   // Определение аварий и предупреждений для отображения на HMI
   // PCV300
   IF "REG_Data".PCV300_Message.Error OR "REG_Data".PCV300_Message.Term_error OR
       "REG_Data".PCV300_Message.Phase_failure OR "REG_Data".PCV300_Status.Error OR
       "REG_Data".PCV300_Status.Fail OR "REG_Master".PCV300_error
   THEN
       "Regs".PCV300_Alarm := true;
   ELSE
       "Regs".PCV300_Alarm := false;
   END_IF;

   IF "REG_Data".PCV300_Message.Warning OR "REG_Data".PCV300_Status.Warning
   THEN
       "Regs".PCV300_Warning := true;
   ELSE
       "Regs".PCV300_Warning := false;
   END_IF;

   // LCV300
   IF "REG_Data".LCV300_Message.Error OR "REG_Data".LCV300_Message.Term_error OR
       "REG_Data".LCV300_Message.Phase_failure OR "REG_Data".LCV300_Status.Error OR
       "REG_Data".LCV300_Status.Fail OR "REG_Master".LCV300_error
   THEN
       "Regs".LCV300_Alarm := true;
   ELSE
       "Regs".LCV300_Alarm := false;
   END_IF;

   IF "REG_Data".LCV300_Message.Warning OR "REG_Data".LCV300_Status.Warning
   THEN
       "Regs".LCV300_Warning := true;
   ELSE
       "Regs".LCV300_Warning := false;
   END_IF;
END_FUNCTION

FUNCTION "Modbus_init" : Void   // FC11, SCL
{ S7_Optimized_Access := 'TRUE' }
VERSION : 0.1
BEGIN
   //************************************************ Регуляторы *****************************************************************
   "PortSettings".Regs."Port" := 258;
   "PortSettings".Regs.Baud := 19200;
   "PortSettings".Regs.Parity := 0;
   "REG_Master".Settings.MB_Addr := 1;
   "REG_Master".State := 10;

   "REG_Master".reqREGmaster := 0;
   "Modbus_Comm_Load_Regs".MODE := 4; // Operating mode 4 = Half duplex (RS485) two-wire mode
   "Modbus_Comm_Load_Regs"(REQ := true,
                           "PORT" := "PortSettings".Regs."Port",
                           BAUD := "PortSettings".Regs.Baud,
                           PARITY := "PortSettings".Regs.Parity,
                           FLOW_CTRL := 0,
                           RTS_ON_DLY := 0,
                           RTS_OFF_DLY := 0,
                           RESP_TO := 1000,
                           DONE => "PortSettings".Regs.Done,
                           ERROR => "PortSettings".Regs.Error,
                           STATUS => "PortSettings".Regs.Status,
                           MB_DB := "Modbus_Master_Regs".MB_DB);

   //************************************************ Передача на верхний уровень **************************************************
   "PortSettings".Up."Port" := 257;
   "PortSettings".Up.Baud := 9600;
   "PortSettings".Up.Parity := 0;

   "Modbus_Comm_Load_Up".MODE := 4; // Operating mode 4 = Half duplex (RS485) two-wire mode
   "Modbus_Comm_Load_Up"(REQ := true,
                         "PORT" := "PortSettings".Up."Port",
                         BAUD := "PortSettings".Up.Baud,
                         PARITY := "PortSettings".Up.Parity,
                         FLOW_CTRL := 0,
                         RTS_ON_DLY := 0,
                         RTS_OFF_DLY := 0,
                         RESP_TO := 1000,
                         DONE => "PortSettings".Up.Done,
                         ERROR => "PortSettings".Up.Error,
                         STATUS => "PortSettings".Up.Status,
                         MB_DB := "Modbus_Slave_Up".MB_DB);

   //************************************************ УВП **************************************************
   "MB_CLIENT_UVP".MB_Unit_ID := 1;
   "MB_CLIENT_UVP".MB_Transaction_ID := 1;
   "UVP_States".Connect_UVP.InterfaceId := 64;
   "UVP_States".Connect_UVP.ID := 1;
   "UVP_States".Connect_UVP.ActiveEstablished := true;
   "UVP_States".Connect_UVP.RemoteAddress.ADDR[1] := 10;
   "UVP_States".Connect_UVP.RemoteAddress.ADDR[2] := 158;
   "UVP_States".Connect_UVP.RemoteAddress.ADDR[3] := 144;
   "UVP_States".Connect_UVP.RemoteAddress.ADDR[4] := 30;
   "UVP_States".Connect_UVP.RemotePort := 502;
END_FUNCTION

FUNCTION "DATA_FC" : Void   // FC14, SCL
{ S7_Optimized_Access := 'TRUE' }
VERSION : 0.1
BEGIN
   // Перекладка данных в DATA

    "DATA".Measuring.PT100_Value := "PT100".Signal_AI.Value;
    "DATA".Measuring.PT100_Circuit := "PT100".Signal_AI.Circuit;
    "DATA".Measuring.TT100_Value := "TT100".Signal_AI.Value;
    "DATA".Measuring.TT100_Circuit := "TT100".Signal_AI.Circuit;
    "DATA".Measuring.LT100_Value := "LT100".Signal_AI.Value;
    "DATA".Measuring.LT100_Circuit := "LT100".Signal_AI.Circuit;
    "DATA".Measuring.AG100_Value := "AG100".Signal_AI.Value;
    "DATA".Measuring. AG100_Circuit := "AG100".Signal_AI.Circuit;
    "DATA".Measuring.PT200_Value := "PT200".Signal_AI.Value;
    "DATA".Measuring.PT200_Circuit := "PT200".Signal_AI.Circuit;
    "DATA".Measuring.TT200_Value := "TT200".Signal_AI.Value;
    "DATA".Measuring.TT200_Circuit := "TT200".Signal_AI.Circuit;
    "DATA".Measuring.LT200_Value := "LT200".Signal_AI.Value;
    "DATA".Measuring.LT200_Circuit := "LT200".Signal_AI.Circuit;
    "DATA".Measuring.AG200_Value := "AG200".Signal_AI.Value;
    "DATA".Measuring.AG200_Circuit := "AG200".Signal_AI.Circuit;
    "DATA".Measuring.TT500_Value := "TT500".Signal_AI.Value;
    "DATA".Measuring.TT500_Circuit := "TT500".Signal_AI.Circuit;
    "DATA".Measuring.PCV300_Pologenie := "REG_Data".PCV300_Pologenie_ok;
    "DATA".Measuring.LCV300_Pologenie := "REG_Data".LCV300_Pologenie_ok;
    //
    "DATA".Measuring.SIKG_Press := "UVP_Data".UVP1_Current_L1.UVP_Press;
    "DATA".Measuring.SIKG_Temp := "UVP_Data".UVP1_Current_L1.UVP_Temp;
    "DATA".Measuring.SIKG_Flow_ru := "UVP_Data".UVP1_Current_L1.UVP_vol_flow_work;
    "DATA".Measuring.SIKG_Flow_stu := "UVP_Data".UVP1_Current_L1.UVP_vol_flow_norm;
    "DATA".Measuring.SIKG_Flow_ru_prev2h := "UVP_Data".UVP1_Cumulative_L1.UVP_Vol_work_prev2h;
    "DATA".Measuring.SIKG_Flow_stu_prev2h := "UVP_Data".UVP1_Cumulative_L1.UVP_Vol_norm_prev2h;
    "DATA".Measuring.SIKG_Flow_ru_prevDay := "UVP_Data".UVP1_Cumulative_L1.UVP_Vol_work_prevDay;
    "DATA".Measuring.SIKG_Flow_stu_prevDay := "UVP_Data".UVP1_Cumulative_L1.UVP_Vol_norm_prevDay;
    "DATA".Measuring.SIKG_total := "UVP_Data".UVP1_Current_L1.UVP_Vol_norm;
    //
    "DATA".Measuring.SIKN_MassFlow := "UVP_Data".UVP1_Current_L2.UVP_Param_vol_flow_work;
    "DATA".Measuring.SIKN_MassFlow_prev2h := "UVP_Data".UVP1_Cumulative_L2.UVP_Param_vol_flow_work_prev2h;
    "DATA".Measuring.SIKN_MassFlow_prevDay := "UVP_Data".UVP1_Cumulative_L2.UVP_Param_vol_flow_work_prevDay;
    "DATA".Measuring.SIKN_total := "UVP_Data".UVP1_Current_L2.UVP_Vol_work;

    // ***************************** СТАТУСЫ УСТРОЙСТВ *********************************
    // Статус XV100
    IF ("DI3".Slot.Pins[6] OR "DATA".Measuring.XV100_no_cmd_close OR "DATA".Measuring.XV100_no_cmd_open) THEN
        "DATA".Measuring.XV100_State := 3; // Авария
    ELSIF ("DI3".Slot.Pins[4] AND NOT "DI3".Slot.Pins[5]) THEN
        "DATA".Measuring.XV100_State := 2; // Открыт
    ELSIF ("DI3".Slot.Pins[5] AND NOT "DI3".Slot.Pins[4]) THEN
        "DATA".Measuring.XV100_State := 1; // Закрыт
    ELSE
        "DATA".Measuring.XV100_State := 0; // Неопределено
    END_IF;

    // Статус обогрева
    IF ("Head".Device.Fail > 0) THEN
        "DATA".Measuring.Head_State := 2; // Авария
    ELSIF ("Head".Device.State = 1) THEN
        "DATA".Measuring.Head_State := 1; // Включен
    ELSIF ("Head".Device.State = 0) THEN
        "DATA".Measuring.Head_State := 0; // Выключен
    END_IF;

    // Статус питания установки
    IF ("Power".Device.Fail > 0) THEN
        "DATA".Measuring.Power_State := 2; // Авария
    ELSIF ("Power".Device.State = 1) THEN
        "DATA".Measuring.Power_State := 1; // Включен
    ELSIF ("Power".Device.State = 0) THEN
        "DATA".Measuring.Power_State := 0; // Выключен
    END_IF;

    "DATA".Measuring.PCV300_Alarm := "Regs".PCV300_Alarm;
    "DATA".Measuring.PCV300_Warning := "Regs".PCV300_Warning;
    "DATA".Measuring.PCV300_Midle := "Regs".PCV300_Midle;
    "DATA".Measuring.PCV300_DIST := "REG_Data".PCV300_Message.Selector_DIST;
    "DATA".Measuring.PCV300_LOCAL := "REG_Data".PCV300_Message.Selector_LOCAL;
    "DATA".Measuring.LCV300_Alarm := "Regs".LCV300_Alarm;
    "DATA".Measuring.LCV300_Warning := "Regs".LCV300_Warning;
    "DATA".Measuring.LCV300_Midle := "Regs".LCV300_Midle;
    "DATA".Measuring.LCV300_DIST := "REG_Data".LCV300_Message.Selector_DIST;
    "DATA".Measuring.LCV300_LOCAL := "REG_Data".LCV300_Message.Selector_LOCAL;
    "DATA".Measuring.LS100 := "DI1".Slot.Pins[0];
    "DATA".Measuring.LS101 := "DI1".Slot.Pins[2];
    "DATA".Measuring.LS200 := "DI1".Slot.Pins[4];
    "DATA".Measuring.LS201 := "DI1".Slot.Pins[6];
    "DATA".Measuring.HS600_Emer_stop := "DI2".Slot.Pins[3];
    "DATA".Measuring.Head_run := "DI2".Slot.Pins[7];
    "DATA".Measuring.Power_run := "DI2".Slot.Pins[6];
    "DATA".Measuring.XV100_open := "DI3".Slot.Pins[4];
    "DATA".Measuring.XV100_close := "DI3".Slot.Pins[5];
    "DATA".Measuring.XV100_fault := "DI3".Slot.Pins[6];
    "DATA".Measuring.Spark := "DO1".Slot.Pins[4];

    "DATA".Measuring.PT100_HH_Alarm := "PT100".Signal_AI.HH_Alarm;
    "DATA".Measuring.PT100_H_Alarm := "PT100".Signal_AI.H_Alarm;
    "DATA".Measuring.PT100_L_Alarm := "PT100".Signal_AI.L_Alarm;
    "DATA".Measuring.PT100_LL_Alarm := "PT100".Signal_AI.LL_Alarm;
    "DATA".Measuring.PT100_Chan_Fail := "PT100".Signal_AI.Chan_Fail;
    "DATA".Measuring.PT100_Sim := "PT100".Signal_AI.Sim_En;

    "DATA".Measuring.TT100_HH_Alarm := "TT100".Signal_AI.HH_Alarm;
    "DATA".Measuring.TT100_H_Alarm := "TT100".Signal_AI.H_Alarm;
    "DATA".Measuring.TT100_L_Alarm := "TT100".Signal_AI.L_Alarm;
    "DATA".Measuring.TT100_LL_Alarm := "TT100".Signal_AI.LL_Alarm;
    "DATA".Measuring.TT100_Chan_Fail := "TT100".Signal_AI.Chan_Fail;
    "DATA".Measuring.TT100_Sim := "TT100".Signal_AI.Sim_En;

    "DATA".Measuring.LT100_HH_Alarm := "LT100".Signal_AI.HH_Alarm;
    "DATA".Measuring.LT100_H_Alarm := "LT100".Signal_AI.H_Alarm;
    "DATA".Measuring.LT100_L_Alarm := "LT100".Signal_AI.L_Alarm;
    "DATA".Measuring.LT100_LL_Alarm := "LT100".Signal_AI.LL_Alarm;
    "DATA".Measuring.LT100_Chan_Fail := "LT100".Signal_AI.Chan_Fail;
    "DATA".Measuring.LT100_Sim := "LT100".Signal_AI.Sim_En;

    "DATA".Measuring.AG100_HH_Alarm := "AG100".Signal_AI.HH_Alarm;
    "DATA".Measuring.AG100_H_Alarm := "AG100".Signal_AI.H_Alarm;
    "DATA".Measuring.AG100_L_Alarm := "AG100".Signal_AI.L_Alarm;
    "DATA".Measuring.AG100_LL_Alarm := "AG100".Signal_AI.LL_Alarm;
    "DATA".Measuring.AG100_Chan_Fail := "AG100".Signal_AI.Chan_Fail;
    "DATA".Measuring.AG100_Sim := "AG100".Signal_AI.Sim_En;

    "DATA".Measuring.PT200_HH_Alarm := "PT200".Signal_AI.HH_Alarm;
    "DATA".Measuring.PT200_H_Alarm := "PT200".Signal_AI.H_Alarm;
    "DATA".Measuring.PT200_L_Alarm := "PT200".Signal_AI.L_Alarm;
    "DATA".Measuring.PT200_LL_Alarm := "PT200".Signal_AI.LL_Alarm;
    "DATA".Measuring.PT200_Chan_Fail := "PT200".Signal_AI.Chan_Fail;
    "DATA".Measuring.PT200_Sim := "PT200".Signal_AI.Sim_En;

    "DATA".Measuring.TT200_HH_Alarm := "TT200".Signal_AI.HH_Alarm;
    "DATA".Measuring.TT200_H_Alarm := "TT200".Signal_AI.H_Alarm;
    "DATA".Measuring.TT200_L_Alarm := "TT200".Signal_AI.L_Alarm;
    "DATA".Measuring.TT200_LL_Alarm := "TT200".Signal_AI.LL_Alarm;
    "DATA".Measuring.TT200_Chan_Fail := "TT200".Signal_AI.Chan_Fail;
    "DATA".Measuring.TT200_Sim := "TT200".Signal_AI.Sim_En;

    "DATA".Measuring.LT200_HH_Alarm := "LT200".Signal_AI.HH_Alarm;
    "DATA".Measuring.LT200_H_Alarm := "LT200".Signal_AI.H_Alarm;
    "DATA".Measuring.LT200_L_Alarm := "LT200".Signal_AI.L_Alarm;
    "DATA".Measuring.LT200_LL_Alarm := "LT200".Signal_AI.LL_Alarm;
    "DATA".Measuring.LT200_Chan_Fail := "LT200".Signal_AI.Chan_Fail;
    "DATA".Measuring.LT200_Sim := "LT200".Signal_AI.Sim_En;

    "DATA".Measuring.AG200_HH_Alarm := "AG200".Signal_AI.HH_Alarm;
    "DATA".Measuring.AG200_H_Alarm := "AG200".Signal_AI.H_Alarm;
    "DATA".Measuring.AG200_L_Alarm := "AG200".Signal_AI.L_Alarm;
    "DATA".Measuring.AG200_LL_Alarm := "AG200".Signal_AI.LL_Alarm;
    "DATA".Measuring.AG200_Chan_Fail := "AG200".Signal_AI.Chan_Fail;
    "DATA".Measuring.AG200_Sim := "AG200".Signal_AI.Sim_En;

    "DATA".Measuring.TT500_HH_Alarm := "TT500".Signal_AI.HH_Alarm;
    "DATA".Measuring.TT500_H_Alarm := "TT500".Signal_AI.H_Alarm;
    "DATA".Measuring.TT500_L_Alarm := "TT500".Signal_AI.L_Alarm;
    "DATA".Measuring.TT500_LL_Alarm := "TT500".Signal_AI.LL_Alarm;
    "DATA".Measuring.TT500_Chan_Fail := "TT500".Signal_AI.Chan_Fail;
    "DATA".Measuring.TT500_Sim := "TT500".Signal_AI.Sim_En;



   // Запись команд из DATA
    "PT100".Signal_AI.Scal_Max_Eu := "DATA".Commands.PT100_Scal_Max_Eu;
    "PT100".Signal_AI.Scal_Min_Eu := "DATA".Commands.PT100_Scal_Min_Eu;
    "PT100".Signal_AI.HH_Lim := "DATA".Commands.PT100_HH_Lim;
    "PT100".Signal_AI.H_Lim := "DATA".Commands.PT100_H_Lim;
    "PT100".Signal_AI.L_Lim := "DATA".Commands.PT100_L_Lim;
    "PT100".Signal_AI.LL_Lim := "DATA".Commands.PT100_LL_Lim;
    "PT100".Signal_AI.Sim_Value := "DATA".Commands.PT100_Sim_Value;

    "TT100".Signal_AI.Scal_Max_Eu := "DATA".Commands.TT100_Scal_Max_Eu;
    "TT100".Signal_AI.Scal_Min_Eu := "DATA".Commands.TT100_Scal_Min_Eu;
    "TT100".Signal_AI.HH_Lim := "DATA".Commands.TT100_HH_Lim;
    "TT100".Signal_AI.H_Lim := "DATA".Commands.TT100_H_Lim;
    "TT100".Signal_AI.L_Lim := "DATA".Commands.TT100_L_Lim;
    "TT100".Signal_AI.LL_Lim := "DATA".Commands.TT100_LL_Lim;
    "TT100".Signal_AI.Sim_Value := "DATA".Commands.TT100_Sim_Value;

    "LT100".Signal_AI.Scal_Max_Eu := "DATA".Commands.LT100_Scal_Max_Eu;
    "LT100".Signal_AI.Scal_Min_Eu := "DATA".Commands.LT100_Scal_Min_Eu;
    "LT100".Signal_AI.HH_Lim := "DATA".Commands.LT100_HH_Lim;
    "LT100".Signal_AI.H_Lim := "DATA".Commands.LT100_H_Lim;
    "LT100".Signal_AI.L_Lim := "DATA".Commands.LT100_L_Lim;
    "LT100".Signal_AI.LL_Lim := "DATA".Commands.LT100_LL_Lim;
    "LT100".Signal_AI.Sim_Value := "DATA".Commands.LT100_Sim_Value;

    "AG100".Signal_AI.Scal_Max_Eu := "DATA".Commands.AG100_Scal_Max_Eu;
    "AG100".Signal_AI.Scal_Min_Eu := "DATA".Commands.AG100_Scal_Min_Eu;
    "AG100".Signal_AI.HH_Lim := "DATA".Commands.AG100_HH_Lim;
    "AG100".Signal_AI.H_Lim := "DATA".Commands.AG100_H_Lim;
    "AG100".Signal_AI.L_Lim := "DATA".Commands.AG100_L_Lim;
    "AG100".Signal_AI.LL_Lim := "DATA".Commands.AG100_LL_Lim;
    "AG100".Signal_AI.Sim_Value := "DATA".Commands.AG100_Sim_Value;

    "PT200".Signal_AI.Scal_Max_Eu := "DATA".Commands.PT200_Scal_Max_Eu;
    "PT200".Signal_AI.Scal_Min_Eu := "DATA".Commands.PT200_Scal_Min_Eu;
    "PT200".Signal_AI.HH_Lim := "DATA".Commands.PT200_HH_Lim;
    "PT200".Signal_AI.H_Lim := "DATA".Commands.PT200_H_Lim;
    "PT200".Signal_AI.L_Lim := "DATA".Commands.PT200_L_Lim;
    "PT200".Signal_AI.LL_Lim := "DATA".Commands.PT200_LL_Lim;
    "PT200".Signal_AI.Sim_Value := "DATA".Commands.PT200_Sim_Value;

    "TT200".Signal_AI.Scal_Max_Eu := "DATA".Commands.TT200_Scal_Max_Eu;
    "TT200".Signal_AI.Scal_Min_Eu := "DATA".Commands.TT200_Scal_Min_Eu;
    "TT200".Signal_AI.HH_Lim := "DATA".Commands.TT200_HH_Lim;
    "TT200".Signal_AI.H_Lim := "DATA".Commands.TT200_H_Lim;
    "TT200".Signal_AI.L_Lim := "DATA".Commands.TT200_L_Lim;
    "TT200".Signal_AI.LL_Lim := "DATA".Commands.TT200_LL_Lim;
    "TT200".Signal_AI.Sim_Value := "DATA".Commands.TT200_Sim_Value;

    "LT200".Signal_AI.Scal_Max_Eu := "DATA".Commands.LT200_Scal_Max_Eu;
    "LT200".Signal_AI.Scal_Min_Eu := "DATA".Commands.LT200_Scal_Min_Eu;
    "LT200".Signal_AI.HH_Lim := "DATA".Commands.LT200_HH_Lim;
    "LT200".Signal_AI.H_Lim := "DATA".Commands.LT200_H_Lim;
    "LT200".Signal_AI.L_Lim := "DATA".Commands.LT200_L_Lim;
    "LT200".Signal_AI.LL_Lim := "DATA".Commands.LT200_LL_Lim;
    "LT200".Signal_AI.Sim_Value := "DATA".Commands.LT200_Sim_Value;

    "AG200".Signal_AI.Scal_Max_Eu := "DATA".Commands.AG200_Scal_Max_Eu;
    "AG200".Signal_AI.Scal_Min_Eu := "DATA".Commands.AG200_Scal_Min_Eu;
    "AG200".Signal_AI.HH_Lim := "DATA".Commands.AG200_HH_Lim;
    "AG200".Signal_AI.H_Lim := "DATA".Commands.AG200_H_Lim;
    "AG200".Signal_AI.L_Lim := "DATA".Commands.AG200_L_Lim;
    "AG200".Signal_AI.LL_Lim := "DATA".Commands.AG200_LL_Lim;
    "AG200".Signal_AI.Sim_Value := "DATA".Commands.AG200_Sim_Value;

    "TT500".Signal_AI.Scal_Max_Eu := "DATA".Commands.TT500_Scal_Max_Eu;
    "TT500".Signal_AI.Scal_Min_Eu := "DATA".Commands.TT500_Scal_Min_Eu;
    "TT500".Signal_AI.HH_Lim := "DATA".Commands.TT500_HH_Lim;
    "TT500".Signal_AI.H_Lim := "DATA".Commands.TT500_H_Lim;
    "TT500".Signal_AI.L_Lim := "DATA".Commands.TT500_L_Lim;
    "TT500".Signal_AI.LL_Lim := "DATA".Commands.TT500_LL_Lim;
    "TT500".Signal_AI.Sim_Value := "DATA".Commands.TT500_Sim_Value;

    "PCV300".Setpoint := "DATA".Commands.PCV300_Setpoint;
    "PCV300".ManualValue := "DATA".Commands.PCV300_ManualValue;
    "PCV300".Retain.CtrlParams.Gain := "DATA".Commands.PCV300_Gain;
    "PCV300".Retain.CtrlParams.Ti := "DATA".Commands.PCV300_Ti;
    "PCV300".Retain.CtrlParams.Td := "DATA".Commands.PCV300_Td;
    "PCV300".Retain.CtrlParams.TdFiltRatio := "DATA".Commands.PCV300_TdFiltRatio;
    "PCV300".Config.OutputUpperLimit := "DATA".Commands.PCV300_OutputUpperLimit;
    "PCV300".Config.OutputLowerLimit := "DATA".Commands.PCV300_OutputLowerLimit;

    "LCV300".Setpoint := "DATA".Commands. LCV300_Setpoint;
    "LCV300".ManualValue := "DATA".Commands. LCV300_ManualValue;
    "LCV300".Retain.CtrlParams.Gain := "DATA".Commands. LCV300_Gain;
    "LCV300".Retain.CtrlParams.Ti := "DATA".Commands. LCV300_Ti;
    "LCV300".Retain.CtrlParams.Td := "DATA".Commands. LCV300_Td;
    "LCV300".Retain.CtrlParams.TdFiltRatio := "DATA".Commands. LCV300_TdFiltRatio;
    "LCV300".Config.OutputUpperLimit := "DATA".Commands. LCV300_OutputUpperLimit;
    "LCV300".Config.OutputLowerLimit := "DATA".Commands. LCV300_OutputLowerLimit;

    "PT100".Signal_AI.HH_Alarm_En := "DATA".Commands.PT100_HH_Alarm_En;
    "PT100".Signal_AI.H_Alarm_En := "DATA".Commands.PT100_H_Alarm_En;
    "PT100".Signal_AI.L_Alarm_En := "DATA".Commands.PT100_L_Alarm_En;
    "PT100".Signal_AI.LL_Alarm_En := "DATA".Commands.PT100_LL_Alarm_En;
    "PT100".Signal_AI.Sim_En := "DATA".Commands.PT100_Sim_En;

    "TT100".Signal_AI.HH_Alarm_En := "DATA".Commands.TT100_HH_Alarm_En;
    "TT100".Signal_AI.H_Alarm_En := "DATA".Commands.TT100_H_Alarm_En;
    "TT100".Signal_AI.L_Alarm_En := "DATA".Commands.TT100_L_Alarm_En;
    "TT100".Signal_AI.LL_Alarm_En := "DATA".Commands.TT100_LL_Alarm_En;
    "TT100".Signal_AI.Sim_En := "DATA".Commands.TT100_Sim_En;

    "LT100".Signal_AI.HH_Alarm_En := "DATA".Commands.LT100_HH_Alarm_En;
    "LT100".Signal_AI.H_Alarm_En := "DATA".Commands.LT100_H_Alarm_En;
    "LT100".Signal_AI.L_Alarm_En := "DATA".Commands.LT100_L_Alarm_En;
    "LT100".Signal_AI.LL_Alarm_En := "DATA".Commands.LT100_LL_Alarm_En;
    "LT100".Signal_AI.Sim_En := "DATA".Commands.LT100_Sim_En;

    "AG100".Signal_AI.HH_Alarm_En := "DATA".Commands.AG100_HH_Alarm_En;
    "AG100".Signal_AI.H_Alarm_En := "DATA".Commands.AG100_H_Alarm_En;
    "AG100".Signal_AI.L_Alarm_En := "DATA".Commands.AG100_L_Alarm_En;
    "AG100".Signal_AI.LL_Alarm_En := "DATA".Commands.AG100_LL_Alarm_En;
    "AG100".Signal_AI.Sim_En := "DATA".Commands.AG100_Sim_En;

    "PT200".Signal_AI.HH_Alarm_En := "DATA".Commands.PT200_HH_Alarm_En;
    "PT200".Signal_AI.H_Alarm_En := "DATA".Commands.PT200_H_Alarm_En;
    "PT200".Signal_AI.L_Alarm_En := "DATA".Commands.PT200_L_Alarm_En;
    "PT200".Signal_AI.LL_Alarm_En := "DATA".Commands.PT200_LL_Alarm_En;
    "PT200".Signal_AI.Sim_En := "DATA".Commands.PT200_Sim_En;

    "TT200".Signal_AI.HH_Alarm_En := "DATA".Commands.TT200_HH_Alarm_En;
    "TT200".Signal_AI.H_Alarm_En := "DATA".Commands.TT200_H_Alarm_En;
    "TT200".Signal_AI.L_Alarm_En := "DATA".Commands.TT200_L_Alarm_En;
    "TT200".Signal_AI.LL_Alarm_En := "DATA".Commands.TT200_LL_Alarm_En;
    "TT200".Signal_AI.Sim_En := "DATA".Commands.TT200_Sim_En;

    "LT200".Signal_AI.HH_Alarm_En := "DATA".Commands.LT200_HH_Alarm_En;
    "LT200".Signal_AI.H_Alarm_En := "DATA".Commands.LT200_H_Alarm_En;
    "LT200".Signal_AI.L_Alarm_En := "DATA".Commands.LT200_L_Alarm_En;
    "LT200".Signal_AI.LL_Alarm_En := "DATA".Commands.LT200_LL_Alarm_En;
    "LT200".Signal_AI.Sim_En := "DATA".Commands.LT200_Sim_En;

    "AG200".Signal_AI.HH_Alarm_En := "DATA".Commands.AG200_HH_Alarm_En;
    "AG200".Signal_AI.H_Alarm_En := "DATA".Commands.AG200_H_Alarm_En;
    "AG200".Signal_AI.L_Alarm_En := "DATA".Commands.AG200_L_Alarm_En;
    "AG200".Signal_AI.LL_Alarm_En := "DATA".Commands.AG200_LL_Alarm_En;
    "AG200".Signal_AI.Sim_En := "DATA".Commands.AG200_Sim_En;

    "TT500".Signal_AI.HH_Alarm_En := "DATA".Commands.TT500_HH_Alarm_En;
    "TT500".Signal_AI.H_Alarm_En := "DATA".Commands.TT500_H_Alarm_En;
    "TT500".Signal_AI.L_Alarm_En := "DATA".Commands.TT500_L_Alarm_En;
    "TT500".Signal_AI.LL_Alarm_En := "DATA".Commands.TT500_LL_Alarm_En;
    "TT500".Signal_AI.Sim_En := "DATA".Commands.TT500_Sim_En;

    "PCV300".ManualEnable := "DATA".Commands.PCV300_ManualEnable;
    "LCV300".ManualEnable := "DATA".Commands.LCV300_ManualEnable;

    // Включение обогрева
    IF "DATA".Commands.Head_cmd_on AND NOT "Head_cmd_on_prev" THEN
        "Head".Device.Cmd_On := 4;
        "DATA".Commands.Head_cmd_on := false;
    END_IF;
    "Head_cmd_on_prev" := "DATA".Commands.Head_cmd_on;

    // Выключение обогрева
    IF "DATA".Commands.Head_cmd_off AND NOT "Head_cmd_off_prev" THEN
        "Head".Device.Cmd_Off := 4;
        "DATA".Commands.Head_cmd_off := false;
    END_IF;
    "Head_cmd_off_prev" := "DATA".Commands.Head_cmd_off;

    // Сброс ошибки обогрева
    IF "DATA".Commands.Head_cmd_reset AND NOT "Power_reset_prev" THEN
        "Head".Device.Cmd_Reset_Error := 4;
        "DATA".Commands.Head_cmd_reset := false;
    END_IF;
    "Head_reset_prev" := "DATA".Commands.Head_cmd_reset;

    // Включение питания
    IF "DATA".Commands.Power_cmd_on AND NOT "Power_cmd_on_prev" THEN
        "Power".Device.Cmd_On := 4;
        "DATA".Commands.Power_cmd_on := false;
    END_IF;
    "Power_cmd_on_prev" := "DATA".Commands.Power_cmd_on;

    // Выключение питания
    IF "DATA".Commands.Power_cmd_off AND NOT "Power_cmd_off_prev" THEN
        "Power".Device.Cmd_Off := 4;
        "DATA".Commands.Power_cmd_off := false;
    END_IF;
    "Power_cmd_off_prev" := "DATA".Commands.Power_cmd_off;

    // Сброс ошибки питания
    IF "DATA".Commands.Power_cmd_reset AND NOT "Power_reset_prev" THEN
        "Power".Device.Cmd_Reset_Error := 4;
        "DATA".Commands.Power_cmd_reset := false;
    END_IF;
    "Power_reset_prev" := "DATA".Commands.Power_cmd_reset;

    IF NOT "Modbus_Comm_Load_Up".DONE THEN
        "Modbus_Comm_Load_Up".MODE := 4; // Operating mode 4 = Half duplex (RS485) two-wire mode
        "Modbus_Comm_Load_Up"(REQ := true,
                              "PORT" := "PortSettings".Up."Port",
                              BAUD := "PortSettings".Up.Baud,
                              PARITY := "PortSettings".Up.Parity,
                              FLOW_CTRL := 0,
                              RTS_ON_DLY := 0,
                              RTS_OFF_DLY := 0,
                              RESP_TO := 1000,
                              DONE => "PortSettings".Up.Done,
                              ERROR => "PortSettings".Up.Error,
                              STATUS => "PortSettings".Up.Status,
                              MB_DB := "Modbus_Slave_Up".MB_DB);
    END_IF;


   // Дополнительно - резервные АИ
    "DATA".AI2_Ch1 := "AI2_Ch1";
    "DATA".AI2_Ch2 := "AI2_Ch2";
    "DATA".AI2_Ch3 := "AI2_Ch3";
    "DATA".AI2_Ch4 := "AI2_Ch4";
    "DATA".AI2_Ch5 := "AI2_Ch5";
    "DATA".AI2_Ch6 := "AI2_Ch6";
    "DATA".AI2_Ch7 := "AI2_Ch7";

   // СИКГ - 2
    "DATA".SIKG2_Press := "UVP_Data".UVP1_Current_L3.UVP_Press;
    "DATA".SIKG2_Temp := "UVP_Data".UVP1_Current_L3.UVP_Temp;
    "DATA".SIKG2_Flow_ru := "UVP_Data".UVP1_Current_L3.UVP_vol_flow_work;
    "DATA".SIKG2_Flow_stu := "UVP_Data".UVP1_Current_L3.UVP_vol_flow_norm;
    "DATA".SIKG2_Flow_ru_prev2h := "UVP_Data".UVP1_Cumulative_L3.UVP_Vol_work_prev2h;
    "DATA".SIKG2_Flow_stu_prev2h := "UVP_Data".UVP1_Cumulative_L3.UVP_Vol_norm_prev2h;
    "DATA".SIKG2_Flow_ru_prevDay := "UVP_Data".UVP1_Cumulative_L3.UVP_Vol_work_prevDay;
    "DATA".SIKG2_Flow_stu_prevDay := "UVP_Data".UVP1_Cumulative_L3.UVP_Vol_norm_prevDay;
    "DATA".SIKG2_total := "UVP_Data".UVP1_Current_L3.UVP_Vol_norm;
   // Объем по уровню
    "DATA".Volume_C1 := "Table".Volume_C1;
    "DATA".Volume_BE := "Table".Volume_BE;
END_FUNCTION